(* Logix 5000 project; controller TBEN_Lx_8IOL_AOI_V0_1 vendor 1 type 14 code 176 rev 32.11; software revision 32.00; part 7 of 11 *)

TYPE Generic_131_Words :
STRUCT
   Data : INT[131];
END_STRUCT
END_TYPE

TYPE Generic_160_SINT :
STRUCT
   DATA : SINT[160];
END_STRUCT
END_TYPE

TYPE Generic_173_Words :
STRUCT
   Data : INT[173];
END_STRUCT
END_TYPE

TYPE Generic_5_Words :
STRUCT
   Data : INT[5];
END_STRUCT
END_TYPE

TYPE IOLRequest :
STRUCT
   Enable_Multiple_Nodes : BOOL;   // Set to 1 to enable multiple nodes
   ApplicationPath : STRING;   // Set Path for following IOL Instructions
   Read : BOOL;   // For internal use to integrate IOLRead and IOWrite with IOLService
   Write : BOOL;   // For internal use to integrate IOLRead and IOWrite with IOLService
   Reset : BOOL;   // For internal use to integrate IOLRead and IOWrite with IOLService
   Done : BOOL;   // For internal use to integrate IOLRead and IOWrite with IOLService
   Error : BOOL;   // For internal use to integrate IOLRead and IOWrite with IOLService
   Slot : INT;   // For internal use to integrate IOLRead and IOWrite with IOLService
   Port : INT;   // For internal use to integrate IOLRead and IOWrite with IOLService
   Index : INT;   // For internal use to integrate IOLRead and IOWrite with IOLService
   SubIndex : INT;   // For internal use to integrate IOLRead and IOWrite with IOLService
   Length : INT;   // For internal use to integrate IOLRead and IOWrite with IOLService
   Handle : INT;   // For internal use to integrate IOLRead and IOWrite with IOLService
   Status : INT;   // For internal use to integrate IOLRead and IOWrite with IOLService
   NextHandle : INT;   // For internal use to integrate IOLRead and IOWrite with IOLService
   ReceiveData : SINT[145];   // For internal use to integrate IOLRead and IOWrite with IOLService
   SendData : SINT[145];   // For internal use to integrate IOLRead and IOWrite with IOLService
   WriteData : DINT;   // For internal use to integrate IOLRead and IOWrite with IOLService
   ActivePath : STRING;   // For internal use to integrate IOLRead and IOWrite with IOLService
END_STRUCT
END_TYPE

TYPE Turck_IOLink_Common_Data :
STRUCT
   Read : BOOL;   // For internal use to integrate IOLRead and IOWrite with IOLService
   Write : BOOL;   // For internal use to integrate IOLRead and IOWrite with IOLService
   Reset : BOOL;   // For internal use to integrate IOLRead and IOWrite with IOLService
   Done : BOOL;   // For internal use to integrate IOLRead and IOWrite with IOLService
   Error : BOOL;   // For internal use to integrate IOLRead and IOWrite with IOLService
   Port_in_Use : SINT;   // Each bit is set to show that a port is in use. If it's not in use the port diagnostics will be disabled so IO-Link can still be used but won't throw a red light if no device plugged
   Port : INT;   // For internal use to integrate IOLRead and IOWrite with IOLService
   Index : INT;   // For internal use to integrate IOLRead and IOWrite with IOLService
   SubIndex : INT;   // For internal use to integrate IOLRead and IOWrite with IOLService
   Length : INT;   // For internal use to integrate IOLRead and IOWrite with IOLService
   TicketNum : INT;   // For internal use to integrate IOLRead and IOWrite with IOLService
   Status : INT;   // For internal use to integrate IOLRead and IOWrite with IOLService
   NextTicketNum : INT;   // For internal use to integrate IOLRead and IOWrite with IOLService
   Process_Input_Data : INT[128];
   Process_Output_Data : INT[128];
   ReceiveData : SINT[255];   // For internal use to integrate IOLRead and IOWrite with IOLService
   SendData : SINT[145];   // For internal use to integrate IOLRead and IOWrite with IOLService
   Vendor_IDs : INT[8];
   Device_IDs : DINT[8];
   WriteData : DINT;
END_STRUCT
END_TYPE

TYPE Universal_IOLink_Info :
STRUCT
   Vendor_Name : STRING;   // Index 16
   Vendor_Text : STRING;   // Index 17
   Product_Name : STRING;   // Index 18
   Product_ID : STRING;   // Index 19
   Product_Text : STRING;   // Index 20
   Serial_Number : STRING;   // Index 21
   Hardware_Revision : STRING;   // Index 22
   Firmware_Revision : STRING;   // Index 23
   Application_Specific_Tag : STRING;   // Index 24
   Function_Tag : STRING;   // Index 25
   Location_Tag : STRING;   // Index 26
   Application_Specific_Tag_Requested : STRING;
END_STRUCT
END_TYPE

ADD_ON_INSTRUCTION IOL_ReadData   (* revision 2.5 Support TBIP, ExecutePrescan, ExecuteEnableInFalse *)
// Revision note:
// V1_0 Initial Release
// V1_1 Automatic data precision detection
// V1_2 Added multiple EIP node support
// V2_5 Support TBIP
// Help:
// IOL_ReadData - used with Turck BL20, BL67, BLC and TBEN IOLink masters to read numeric data from IOLink devices.  Use in conjuction with IOLService AOI which processes all IOL read and write requests.
// Status	Description
// 0	Operation completed successfully
// 	Status = 100 - 102, Ethernet IP MSG instruction errors - check communication parameters
// 100	IOL_SendMSG completed with error, check communication parameters
// 101	IOL_RecevieMSG completed with error, check communication parameters
// 110	IOL_Service Retry Limit exceeded
// 111	Slot specified not an IOLink master
// 	Status = 1000 to 1255, no response from device, connection error
// 1016	Device not connected or Port not configured as IOLink port
// 	Status = 2000 to 2255,  device response indicates error
// 2000	Device error, no details
// 2017	Device error, Index not available
// 2018	Device error, Subindex not available
// 2032	Device error, Service temporarily not available
// 2033	Device error, Service temporarily not available - local control
// 2034	Device error, Service temporarily not available - device control
// 2035	Device error, Index not writeable
// 2048	Device error, Parameter value out of range
// 2049	Device error, Parameter value above limit
// 2050	Device error, Parameter value below limit
// 2051	Device error, Parameter value length overrun (check IOLWrite precision/string length)
// 2052	Device error, Parameter value length underrun (check IOLWrite precision/string length)
// 2053	Device error, Function not available
// 2054	Device error, Function temporarily not available
// 2064	Device error, Parameter set invalid
// 2065	Device error, Inconsistent parameter set
// 2130	Device error, Application not ready
// 	Status = 3000 to 3255,   device response indicates vendor specific error
// 3000	Vendor specific error, no details
// 3001	Vendor specific error, vendor specific error number
// 3255	Vendor specific error, vendor specific error number
// 	Status = 7000 to 7255,  IOL-M Error Codes
// 7000	Unexpected write request instead of read request
// 7001	Decode error
// 7002	Port occupied by another task
// 	Status = 8000 to 8255,  IOL-M Error Codes
// 8000	Timeout when IOL-Ds or IOL-M ports are busy
// 8001	IOL Index out of range
// 8002	Port address greater than maximum
// 8003	Port function not supported
VAR_OUTPUT
   Done : BOOL; {access Read Only, visible}   // IOLRead completed successfully
   Error : BOOL; {access Read Only, visible}   // IOLRead completed with error, check status
   Pending : BOOL; {access Read Only, visible}   // IOLRead waiting to be processed
   Active : BOOL; {access Read Only, visible}   // IOLRead in progress
END_VAR
VAR_IN_OUT
   Common_Data : IOLRequest; {required}   // Shared IOL Data Area - must be identical on all requests
END_VAR
VAR_OUTPUT
   DoneCount : DINT; {access Read Only, visible}   // Number of operations completed successfully
   ErrorCount : DINT; {access Read Only, visible}   // Number of operations competed with error
   Status : INT; {access Read Only, visible}   // Status of last IOLRead
END_VAR
VAR_INPUT
   Read : BOOL;   // Rising edge triggers IOLink Read
   Read_Continuous : BOOL;   // Set to trigger IOLink Read repeatedly
   Slot : INT; {visible}   // IOLink Master slot number
   Port : INT; {visible}   // IOLink Master Port number, 1,2,3 or 4
   Index : INT; {visible}   // IOL Index number
   SubIndex : INT; {visible}   // IOL Subindex number
END_VAR
VAR_OUTPUT
   ReadData : DINT; {access Read Only, required}   // Data returned from IOLink device
END_VAR
VAR_INPUT
   R_8_Bit : BOOL;   // Indicates data received is 8 bit precision
   R_16_Bit : BOOL;   // Indicates data received is 16 bit precision
   R_32_Bit : BOOL;   // Indicates data received is 32 bit precision
   R_Sign_Extend : BOOL;   // Set to extend 8/16 bit precision data sign bit
   R_Swap_16 : BOOL;   // 16-bit AB->BA, 32-bit ABCD->BADC
   R_Swap_32 : BOOL;   // 32-bit ABCD->DCBA
   R_Swap_All : BOOL;   // 32-bit ABCD->CDBA
END_VAR
VAR
   MyHandle : INT;
   StartupDone : BOOL; {access None}
   Pending_or_Active : BOOL; {access None}
   Read_ONS : BOOL; {access None}
   StartupCount : DINT; {access None}
   ReadSignBit : DINT; {access None}
   ReadRequest : BOOL; {access None}
END_VAR

ROUTINE EnableInFalse   (* ladder *)
END_ROUTINE

ROUTINE Logic   (* ladder *)
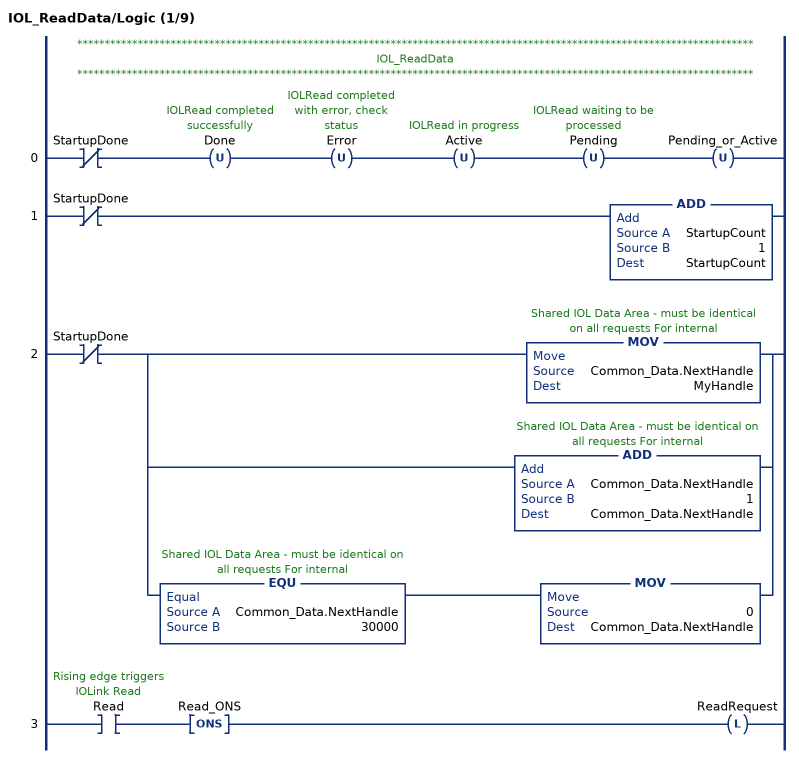
   // ***************************************************************************************************************************
   // IOL_ReadData
   // ***************************************************************************************************************************
   0: XIO(StartupDone)OTU(Done)OTU(Error)OTU(Active)OTU(Pending)OTU(Pending_or_Active);
   1: XIO(StartupDone)ADD(StartupCount,1,StartupCount);
   2: XIO(StartupDone)[MOV(Common_Data.NextHandle,MyHandle) ,ADD(Common_Data.NextHandle,1,Common_Data.NextHandle) ,EQU(Common_Data.NextHandle,30000) MOV(0,Common_Data.NextHandle) ];
   3: XIC(Read)ONS(Read_ONS)OTL(ReadRequest);
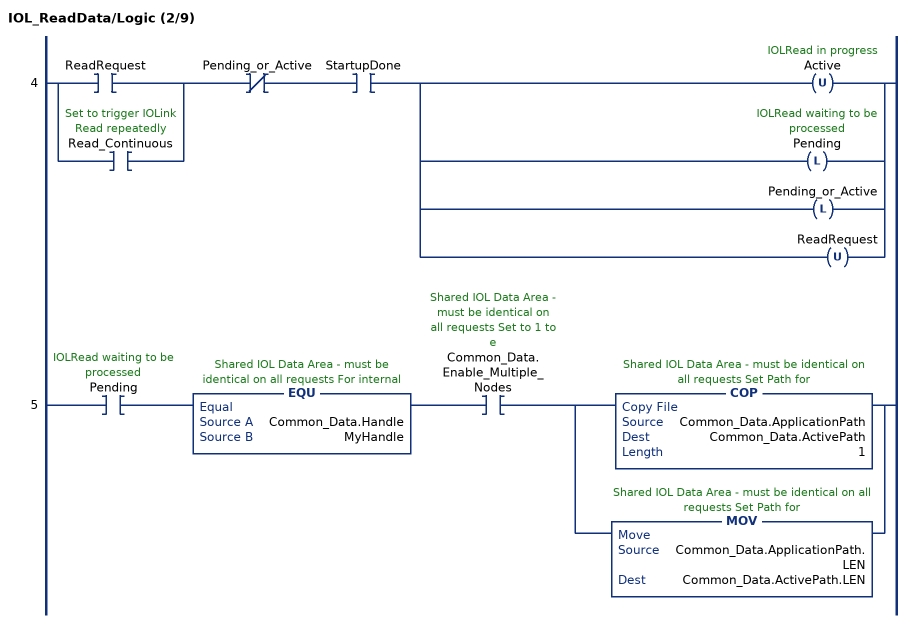
   4: [XIC(ReadRequest) ,XIC(Read_Continuous) ]XIO(Pending_or_Active)XIC(StartupDone)[OTU(Active) ,OTL(Pending) ,OTL(Pending_or_Active) ,OTU(ReadRequest) ];
   5: XIC(Pending)EQU(Common_Data.Handle,MyHandle)XIC(Common_Data.Enable_Multiple_Nodes)[COP(Common_Data.ApplicationPath,Common_Data.ActivePath,1) ,MOV(Common_Data.ApplicationPath.LEN,Common_Data.ActivePath.LEN) ];
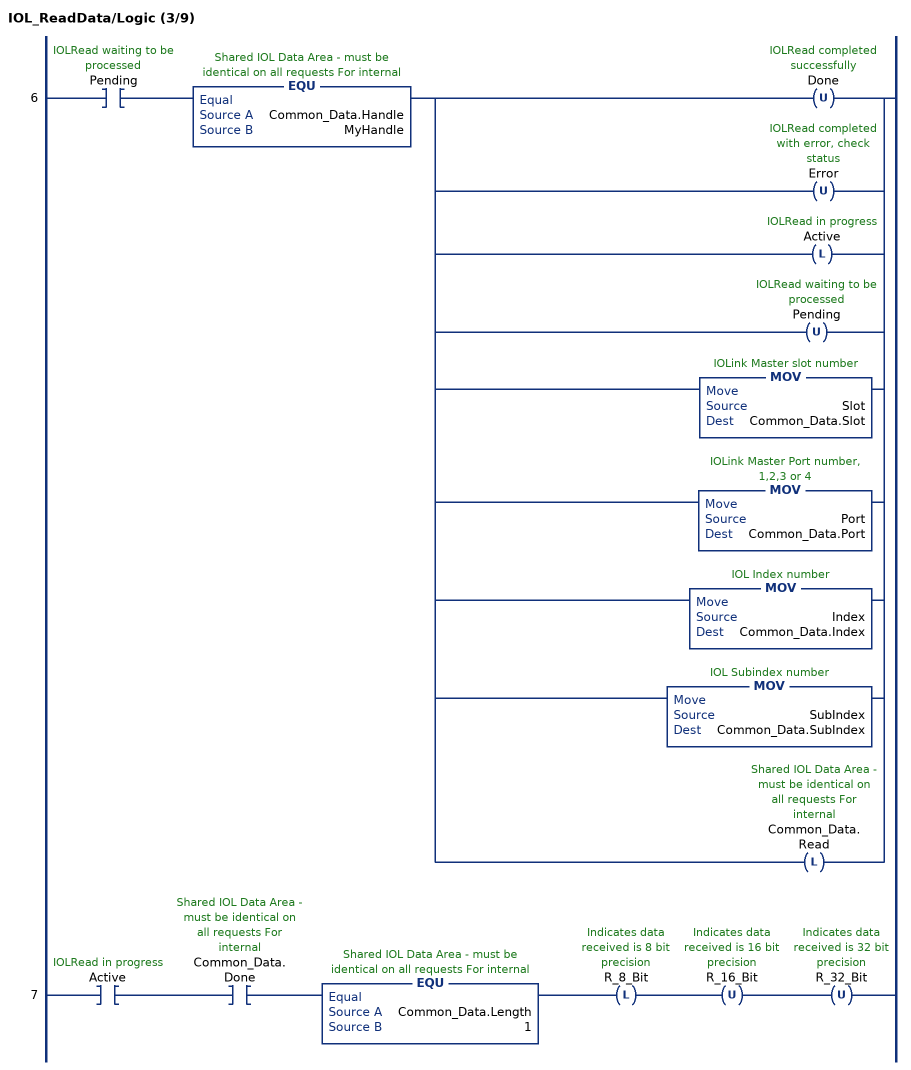
   6: XIC(Pending)EQU(Common_Data.Handle,MyHandle)[OTU(Done) ,OTU(Error) ,OTL(Active) ,OTU(Pending) ,MOV(Slot,Common_Data.Slot) ,MOV(Port,Common_Data.Port) ,MOV(Index,Common_Data.Index) ,MOV(SubIndex,Common_Data.SubIndex) ,OTL(Common_Data.Read) ];
   7: XIC(Active)XIC(Common_Data.Done)EQU(Common_Data.Length,1)OTL(R_8_Bit)OTU(R_16_Bit)OTU(R_32_Bit);
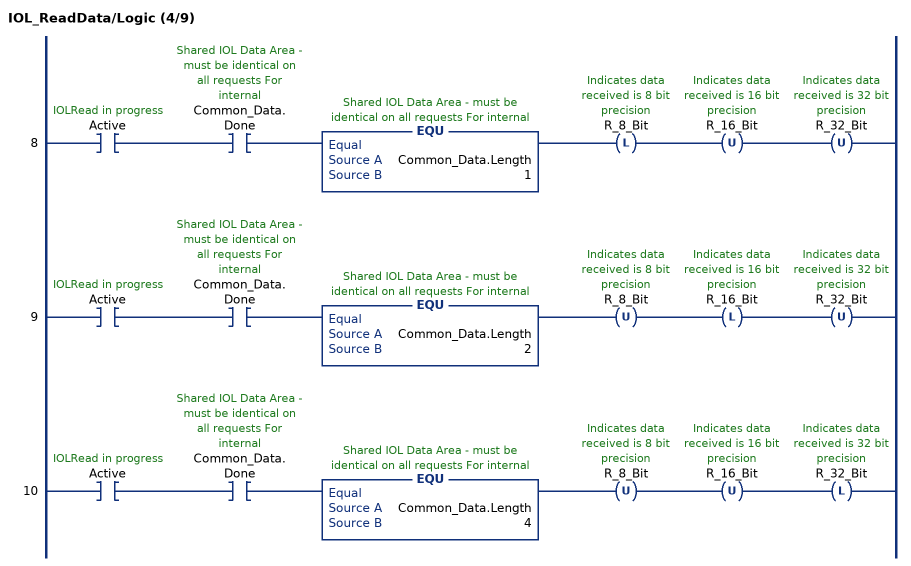
   8: XIC(Active)XIC(Common_Data.Done)EQU(Common_Data.Length,1)OTL(R_8_Bit)OTU(R_16_Bit)OTU(R_32_Bit);
   9: XIC(Active)XIC(Common_Data.Done)EQU(Common_Data.Length,2)OTU(R_8_Bit)OTL(R_16_Bit)OTU(R_32_Bit);
   10: XIC(Active)XIC(Common_Data.Done)EQU(Common_Data.Length,4)OTU(R_8_Bit)OTU(R_16_Bit)OTL(R_32_Bit);
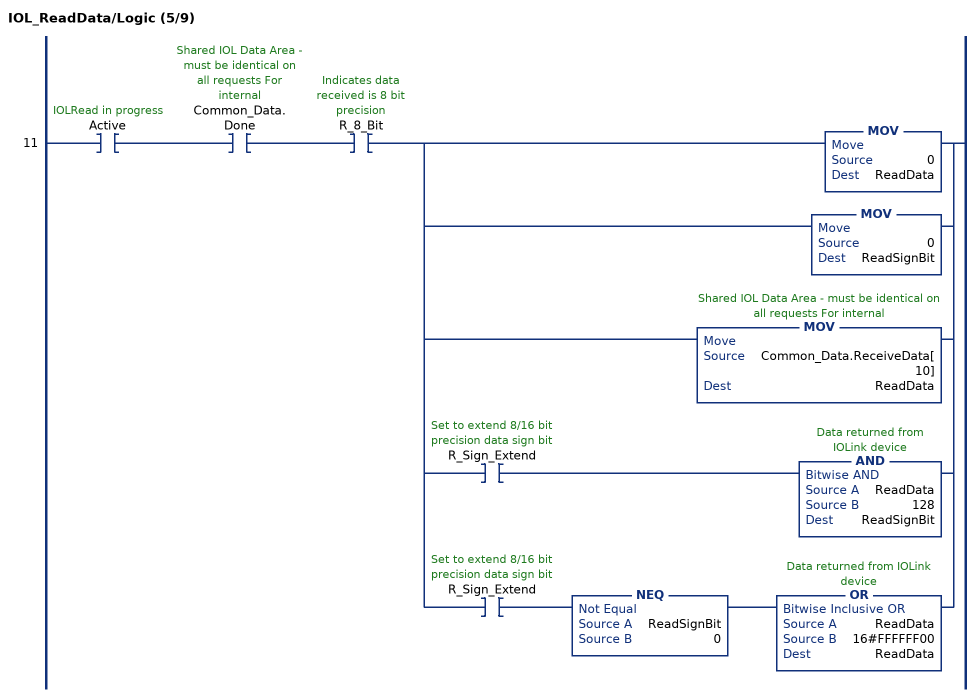
   11: XIC(Active)XIC(Common_Data.Done)XIC(R_8_Bit)[MOV(0,ReadData) ,MOV(0,ReadSignBit) ,MOV(Common_Data.ReceiveData[10],ReadData) ,XIC(R_Sign_Extend) AND(ReadData,128,ReadSignBit) ,XIC(R_Sign_Extend) NEQ(ReadSignBit,0) OR(ReadData,16#FFFFFF00,ReadData) ];
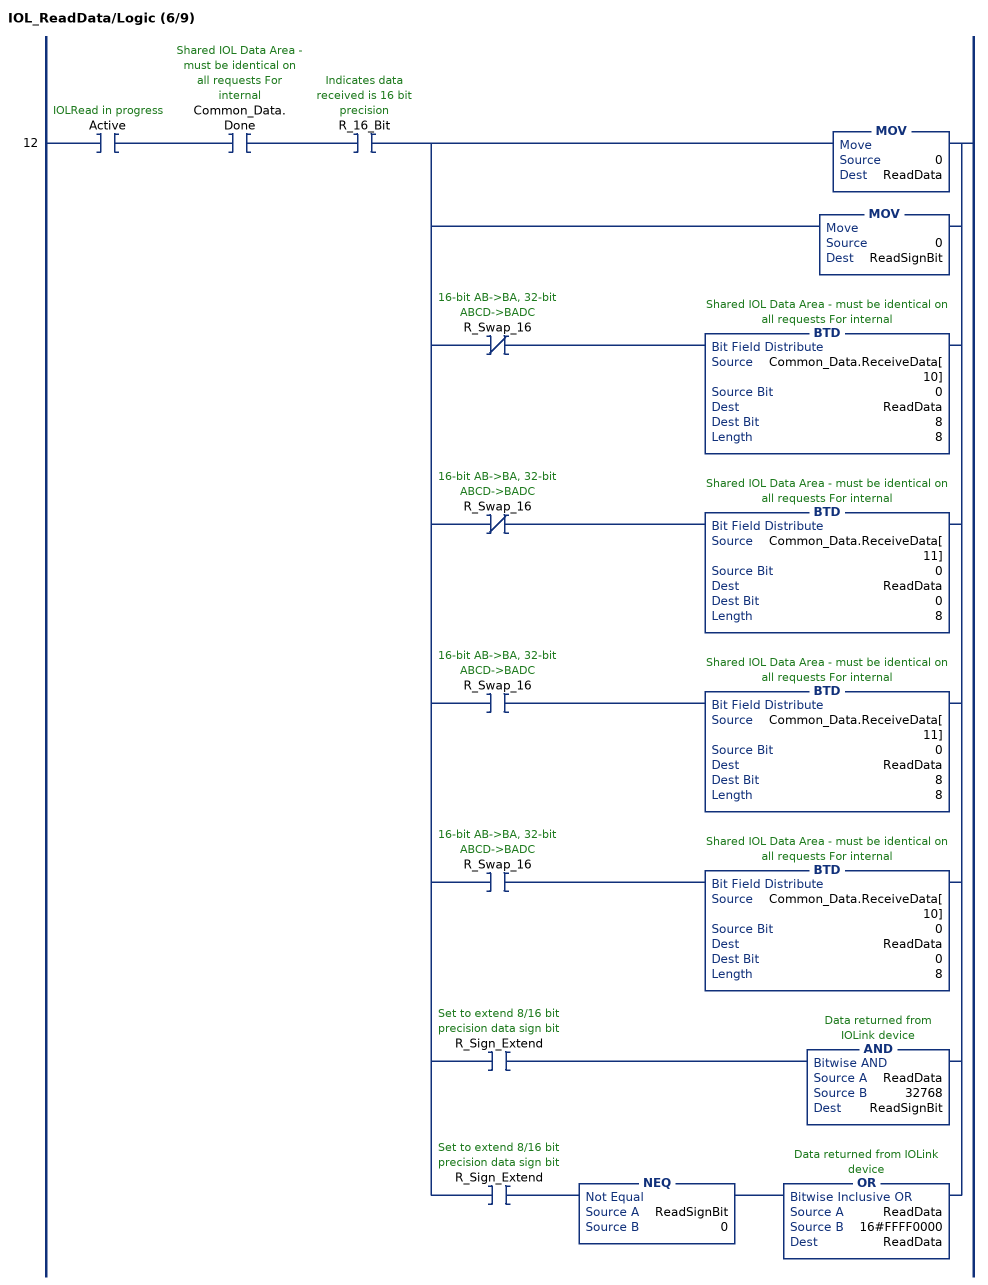
   12: XIC(Active)XIC(Common_Data.Done)XIC(R_16_Bit)[MOV(0,ReadData) ,MOV(0,ReadSignBit) ,XIO(R_Swap_16) BTD(Common_Data.ReceiveData[10],0,ReadData,8,8) ,XIO(R_Swap_16) BTD(Common_Data.ReceiveData[11],0,ReadData,0,8) ,XIC(R_Swap_16) BTD(Common_Data.ReceiveData[11],0,ReadData,8,8) ,XIC(R_Swap_16) BTD(Common_Data.ReceiveData[10],0,ReadData,0,8) ,XIC(R_Sign_Extend) AND(ReadData,32768,ReadSignBit) ,XIC(R_Sign_Extend) NEQ(ReadSignBit,0) OR(ReadData,16#FFFF0000,ReadData) ];
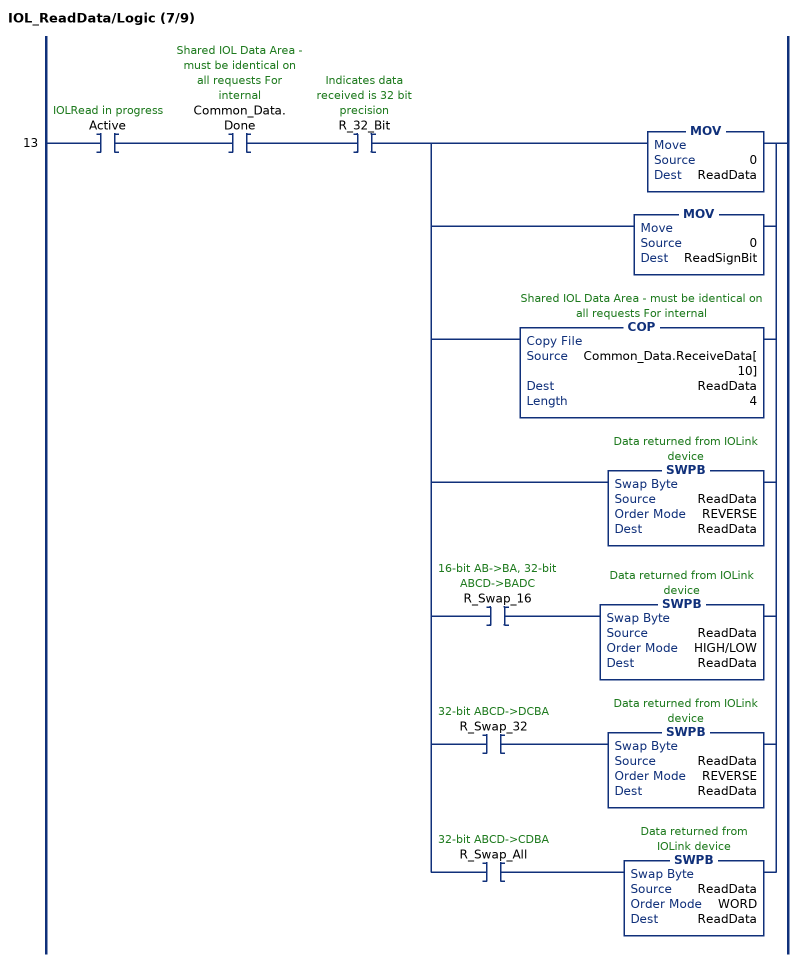
   13: XIC(Active)XIC(Common_Data.Done)XIC(R_32_Bit)[MOV(0,ReadData) ,MOV(0,ReadSignBit) ,COP(Common_Data.ReceiveData[10],ReadData,4) ,SWPB(ReadData,REVERSE,ReadData) ,XIC(R_Swap_16) SWPB(ReadData,HIGH/LOW,ReadData) ,XIC(R_Swap_32) SWPB(ReadData,REVERSE,ReadData) ,XIC(R_Swap_All) SWPB(ReadData,WORD,ReadData) ];
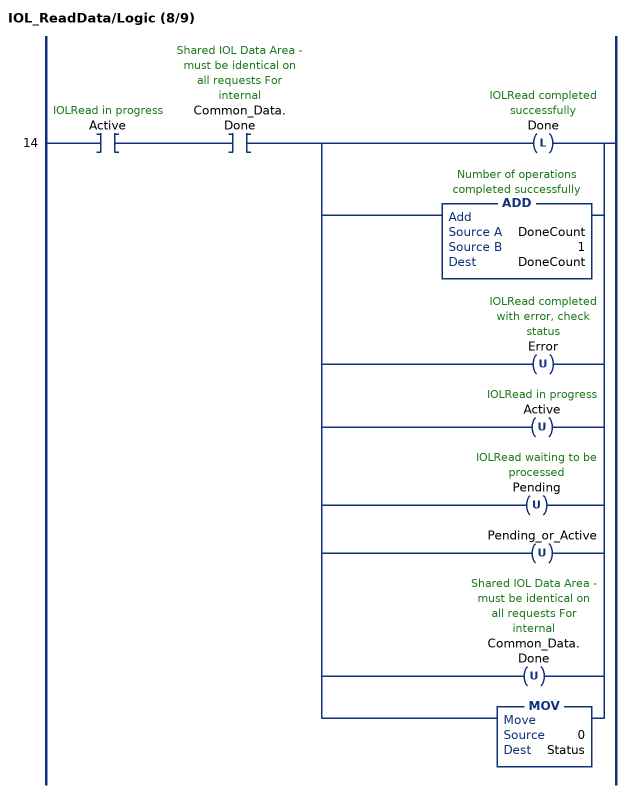
   14: XIC(Active)XIC(Common_Data.Done)[OTL(Done) ,ADD(DoneCount,1,DoneCount) ,OTU(Error) ,OTU(Active) ,OTU(Pending) ,OTU(Pending_or_Active) ,OTU(Common_Data.Done) ,MOV(0,Status) ];
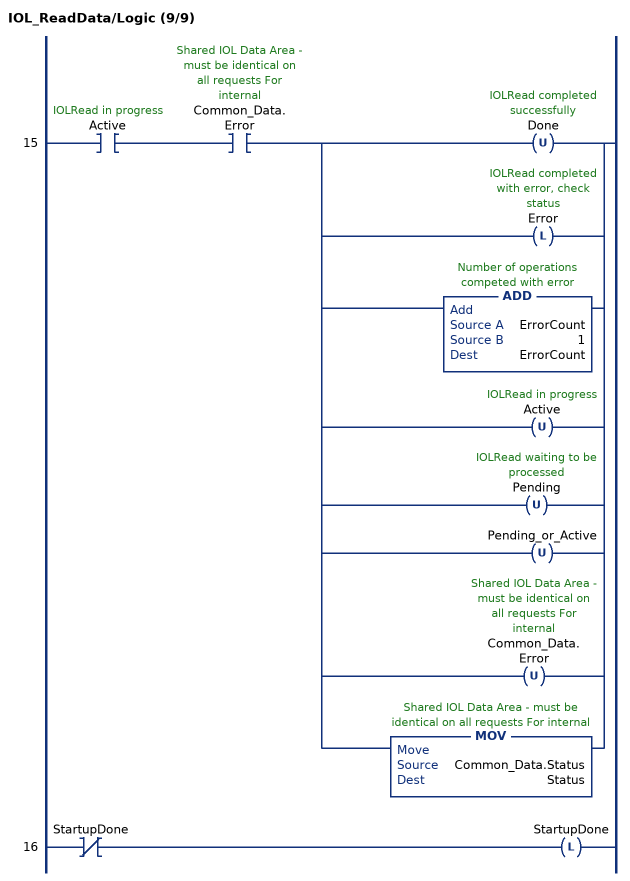
   15: XIC(Active)XIC(Common_Data.Error)[OTU(Done) ,OTL(Error) ,ADD(ErrorCount,1,ErrorCount) ,OTU(Active) ,OTU(Pending) ,OTU(Pending_or_Active) ,OTU(Common_Data.Error) ,MOV(Common_Data.Status,Status) ];
   16: XIO(StartupDone)OTL(StartupDone);
END_ROUTINE

ROUTINE Prescan   (* ladder *)
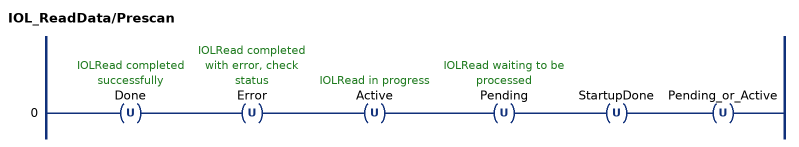
   0: OTU(Done)OTU(Error)OTU(Active)OTU(Pending)OTU(StartupDone)OTU(Pending_or_Active);
END_ROUTINE
END_ADD_ON_INSTRUCTION

ADD_ON_INSTRUCTION IOLService_ISDU   (* revision 1.0 Initial Release, ExecutePrescan *)
// Replace DSID with ISDU in Turck IOLC AOI interface
// KH 6/19/2023
// Revision note:
// V1_0 Initial Release
// Help:
// IOL_Service - used with Turck BL20, BL67, BLC and TBEN IOLink masters to process requests from IOL_ReadString, IOL_WriteString, IOL_ReadData and IOL_WriteData AOI's.
// Status	Description
// 0	Operation completed successfully
// 	Status = 100 - 102, Ethernet IP MSG instruction errors - check communication parameters
// 100	IOL_SendMSG completed with error, check communication parameters
// 101	IOL_RecevieMSG completed with error, check communication parameters
// 110	IOL_Service Retry Limit exceeded
// 111	Slot specified not an IOLink master
// 	Status = 1000 to 1255, no response from device, connection error
// 1016	Device not connected or Port not configured as IOLink port
// 	Status = 2000 to 2255,  device response indicates error
// 2000	Device error, no details
// 2017	Device error, Index not available
// 2018	Device error, Subindex not available
// 2032	Device error, Service temporarily not available
// 2033	Device error, Service temporarily not available - local control
// 2034	Device error, Service temporarily not available - device control
// 2035	Device error, Index not writeable
// 2048	Device error, Parameter value out of range
// 2049	Device error, Parameter value above limit
// 2050	Device error, Parameter value below limit
// 2051	Device error, Parameter value length overrun (check IOLWrite precision/string length)
// 2052	Device error, Parameter value length underrun (check IOLWrite precision/string length)
// 2053	Device error, Function not available
// 2054	Device error, Function temporarily not available
// 2064	Device error, Parameter set invalid
// 2065	Device error, Inconsistent parameter set
// 2130	Device error, Application not ready
// 	Status = 3000 to 3255,   device response indicates vendor specific error
// 3000	Vendor specific error, no details
// 3001	Vendor specific error, vendor specific error number
// 3255	Vendor specific error, vendor specific error number
// 	Status = 7000 to 7255,  IOL-M Error Codes
// 7000	Unexpected write request instead of read request
// 7001	Decode error
// 7002	Port occupied by another task
// 	Status = 8000 to 8255,  IOL-M Error Codes
// 8000	Timeout when IOL-Ds or IOL-M ports are busy
// 8001	IOL Index out of range
// 8002	Port address greater than maximum
// 8003	Port function not supported
VAR_IN_OUT
   Common_Data : Turck_IOLink_Common_Data; {required}
        .SendData[1]   // For internal use to integrate IOLRead and IOLWrite with IOLService
   IOL_Read_MSG : MESSAGE; {required}
   IOL_Write_MSG : MESSAGE; {required}
   Process_Input_Data : Generic_173_Words; {required}
   Process_Output_Data : Generic_131_Words; {required}
END_VAR
VAR
   IOLReadActive : BOOL;
   IOLWriteActive : BOOL;
   RetryCount : DINT;
   IOL_Error_Count : DINT; {access None}
   IOLReset_ONS : BOOL; {access None}
   ER1 : BOOL; {access None}
   ER2 : BOOL; {access None}
   tempReceiveData : SINT[255]; {access None}
   Generate_Status : BOOL; {access None}
   ABS_RD_0 : INT; {access None}
   ABS_RD_1 : INT; {access None}
   ABS_RD_2 : INT; {access None}
   ABS_RD_3 : INT; {access None}
   tempSendData : SINT[145]; {access None}
   IOL_READ_Request : BOOL; {access None}
   IOL_WRITE_Request : BOOL; {access None}
   StartupDone : BOOL; {access None}
   Done : BOOL; {access None}
   Error : BOOL; {access None}
   Active : BOOL; {access None}
   Pending : BOOL; {access None}
   Pending_or_Active : BOOL; {access None}
   StartupCount : SINT; {access None}
   DoneCount : SINT; {access None}
   MyTicketNum : INT; {access None}
   Update_Data : BOOL; {access None}
   Read_ONS : BOOL; {access None}
   ReadRequest : BOOL; {access None}
   Prev_Input_Data_Valids : INT; {access None}
   Status : DINT; {access None}
   ErrorCount : DINT; {access None}
   PIDV_Delay : TIMER := (PRE := 1000); {access None}
END_VAR

ROUTINE Logic   (* ladder *)
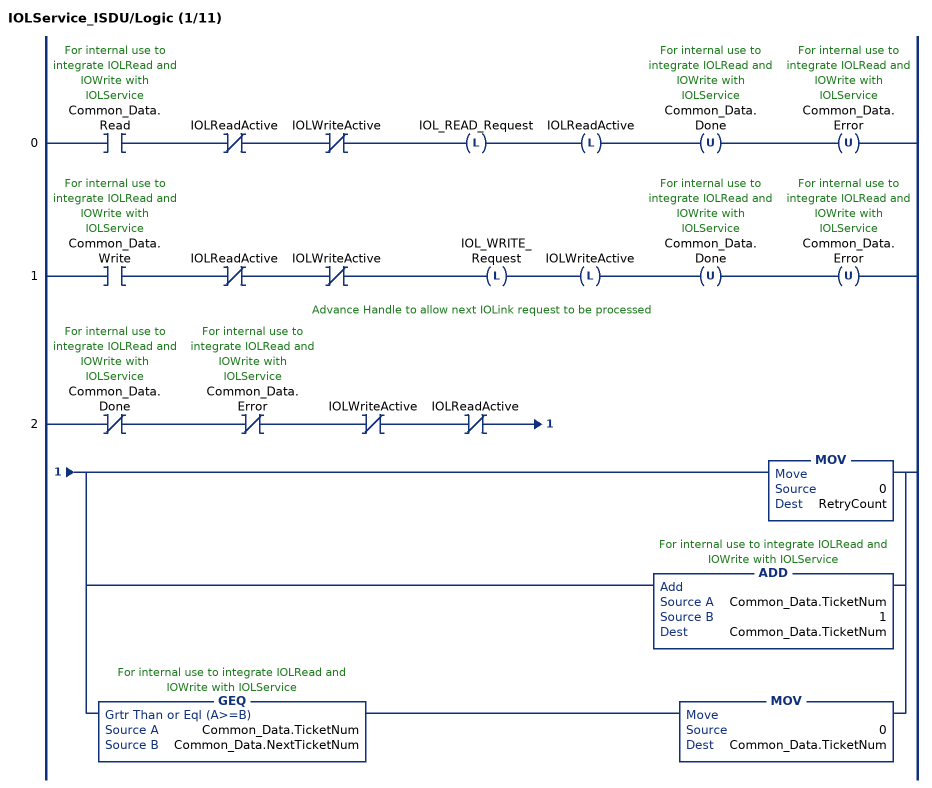
   0: XIC(Common_Data.Read)XIO(IOLReadActive)XIO(IOLWriteActive)OTL(IOL_READ_Request)OTL(IOLReadActive)OTU(Common_Data.Done)OTU(Common_Data.Error);
   1: XIC(Common_Data.Write)XIO(IOLReadActive)XIO(IOLWriteActive)OTL(IOL_WRITE_Request)OTL(IOLWriteActive)OTU(Common_Data.Done)OTU(Common_Data.Error);
   // Advance Handle to allow next IOLink request to be processed
   2: XIO(Common_Data.Done)XIO(Common_Data.Error)XIO(IOLWriteActive)XIO(IOLReadActive)[MOV(0,RetryCount) ,ADD(Common_Data.TicketNum,1,Common_Data.TicketNum) ,GEQ(Common_Data.TicketNum,Common_Data.NextTicketNum) MOV(0,Common_Data.TicketNum) ];
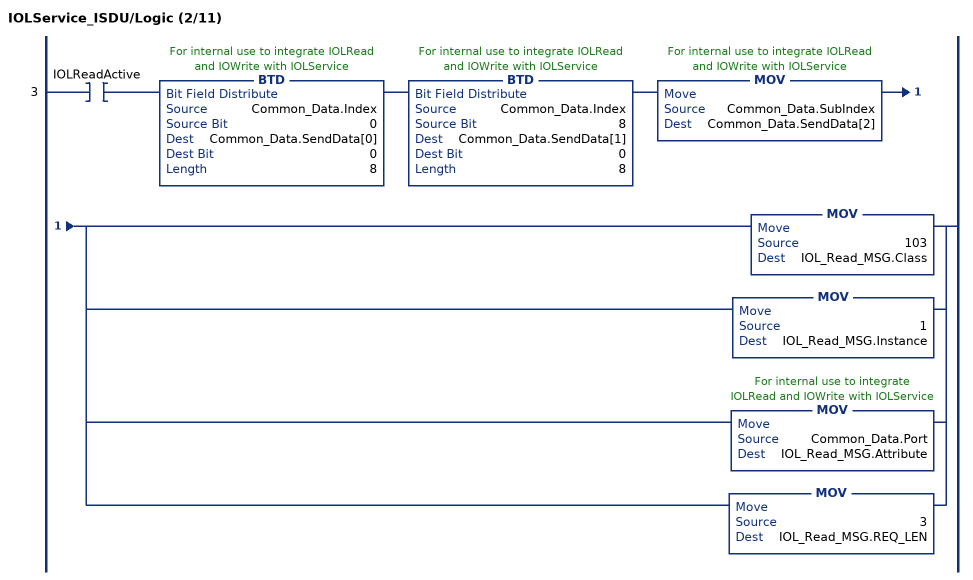
   3: XIC(IOLReadActive)BTD(Common_Data.Index,0,Common_Data.SendData[0],0,8)BTD(Common_Data.Index,8,Common_Data.SendData[1],0,8)MOV(Common_Data.SubIndex,Common_Data.SendData[2])[MOV(103,IOL_Read_MSG.Class) ,MOV(1,IOL_Read_MSG.Instance) ,MOV(Common_Data.Port,IOL_Read_MSG.Attribute) ,MOV(3,IOL_Read_MSG.REQ_LEN) ];
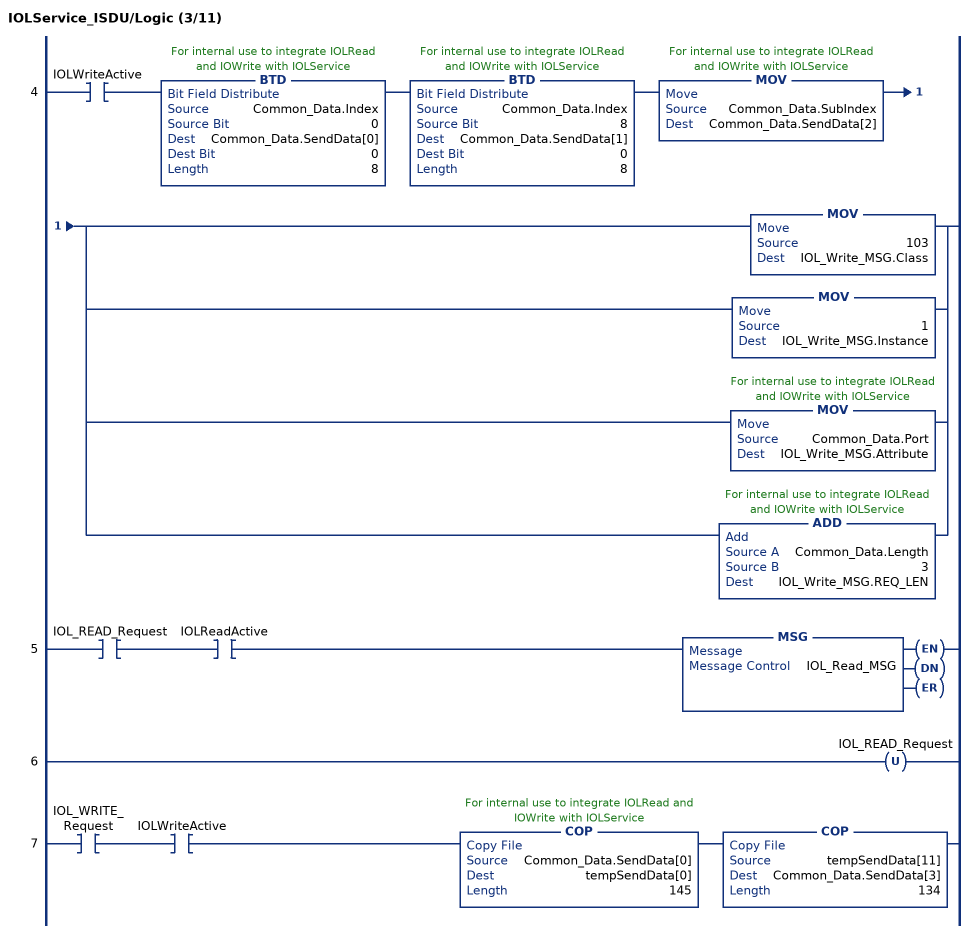
   4: XIC(IOLWriteActive)BTD(Common_Data.Index,0,Common_Data.SendData[0],0,8)BTD(Common_Data.Index,8,Common_Data.SendData[1],0,8)MOV(Common_Data.SubIndex,Common_Data.SendData[2])[MOV(103,IOL_Write_MSG.Class) ,MOV(1,IOL_Write_MSG.Instance) ,MOV(Common_Data.Port,IOL_Write_MSG.Attribute) ,ADD(Common_Data.Length,3,IOL_Write_MSG.REQ_LEN) ];
   5: XIC(IOL_READ_Request)XIC(IOLReadActive)MSG(IOL_Read_MSG);
   6: OTU(IOL_READ_Request);
   7: XIC(IOL_WRITE_Request)XIC(IOLWriteActive)COP(Common_Data.SendData[0],tempSendData[0],145)COP(tempSendData[11],Common_Data.SendData[3],134);
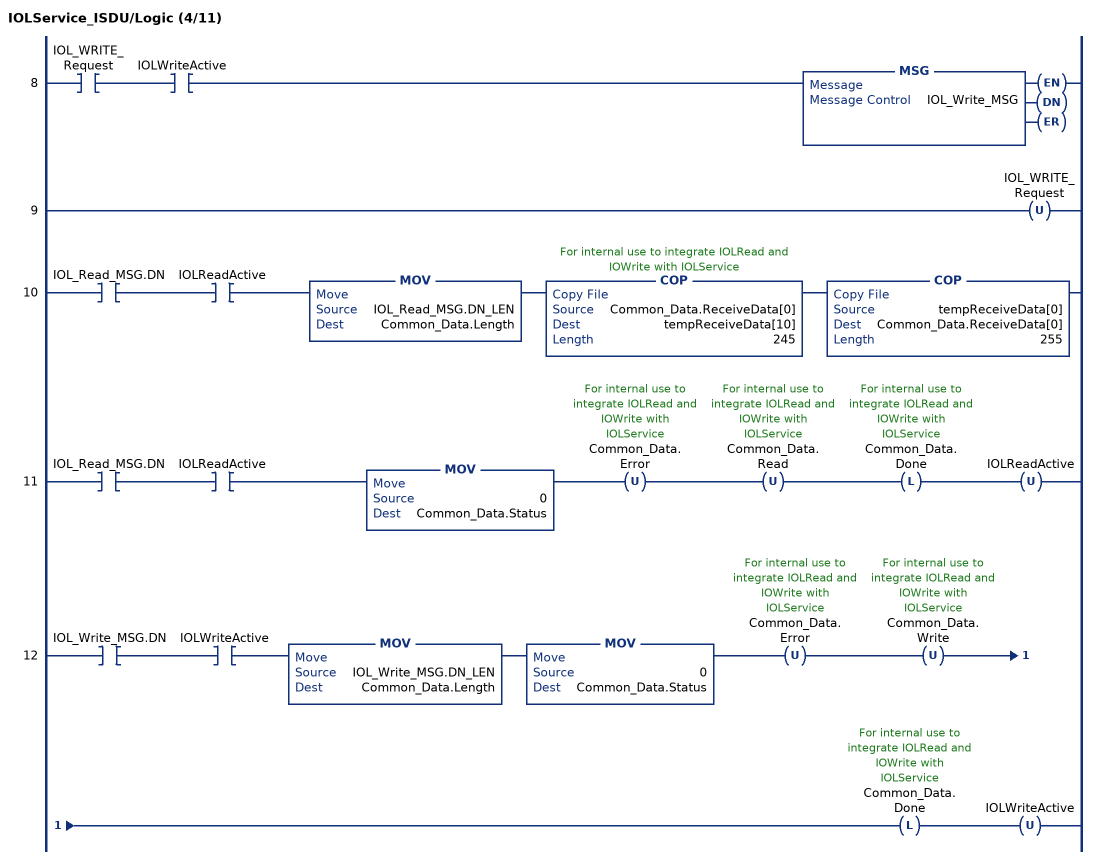
   8: XIC(IOL_WRITE_Request)XIC(IOLWriteActive)MSG(IOL_Write_MSG);
   9: OTU(IOL_WRITE_Request);
   10: XIC(IOL_Read_MSG.DN)XIC(IOLReadActive)MOV(IOL_Read_MSG.DN_LEN,Common_Data.Length)COP(Common_Data.ReceiveData[0],tempReceiveData[10],245)COP(tempReceiveData[0],Common_Data.ReceiveData[0],255);
   11: XIC(IOL_Read_MSG.DN)XIC(IOLReadActive)MOV(0,Common_Data.Status)OTU(Common_Data.Error)OTU(Common_Data.Read)OTL(Common_Data.Done)OTU(IOLReadActive);
   12: XIC(IOL_Write_MSG.DN)XIC(IOLWriteActive)MOV(IOL_Write_MSG.DN_LEN,Common_Data.Length)MOV(0,Common_Data.Status)OTU(Common_Data.Error)OTU(Common_Data.Write)OTL(Common_Data.Done)OTU(IOLWriteActive);
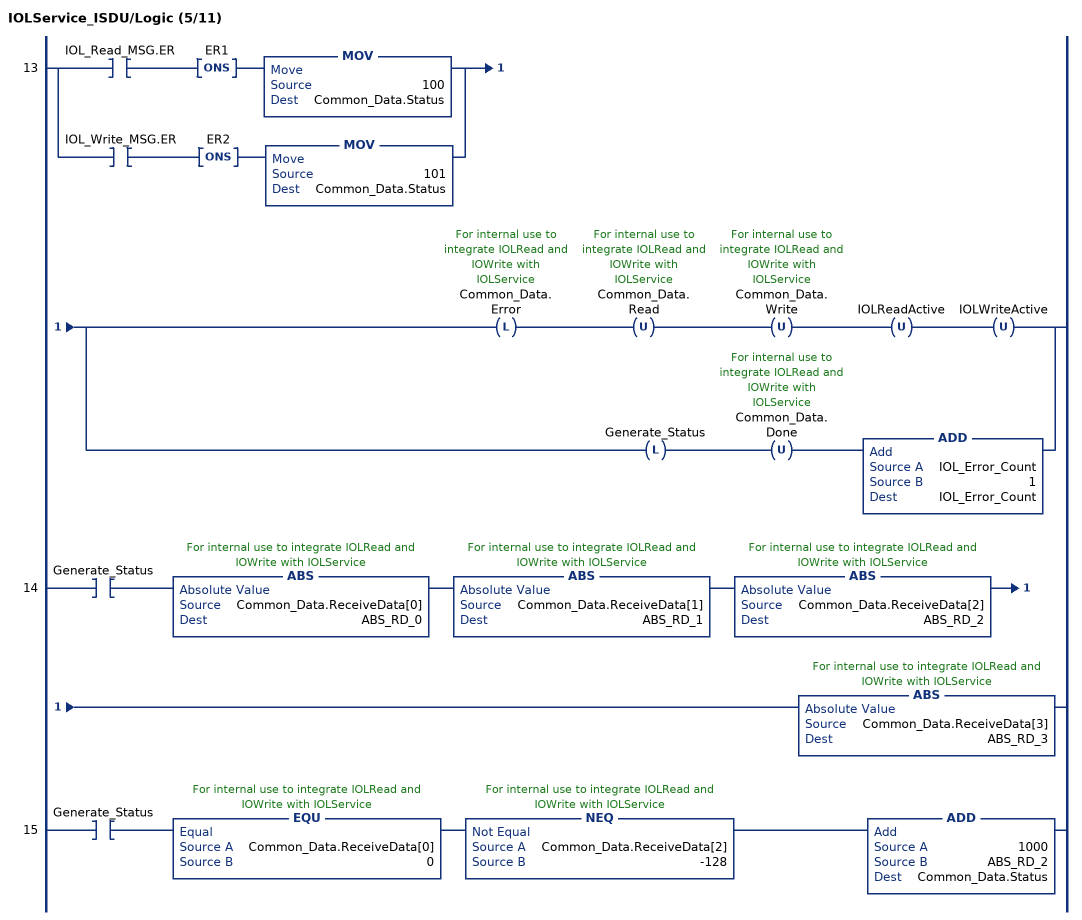
   13: [XIC(IOL_Read_MSG.ER) ONS(ER1) MOV(100,Common_Data.Status) ,XIC(IOL_Write_MSG.ER) ONS(ER2) MOV(101,Common_Data.Status) ][OTL(Common_Data.Error) OTU(Common_Data.Read) OTU(Common_Data.Write) OTU(IOLReadActive) OTU(IOLWriteActive) ,OTL(Generate_Status) OTU(Common_Data.Done) ADD(IOL_Error_Count,1,IOL_Error_Count) ];
   14: XIC(Generate_Status)ABS(Common_Data.ReceiveData[0],ABS_RD_0)ABS(Common_Data.ReceiveData[1],ABS_RD_1)ABS(Common_Data.ReceiveData[2],ABS_RD_2)ABS(Common_Data.ReceiveData[3],ABS_RD_3);
   15: XIC(Generate_Status)EQU(Common_Data.ReceiveData[0],0)NEQ(Common_Data.ReceiveData[2],-128)ADD(1000,ABS_RD_2,Common_Data.Status);
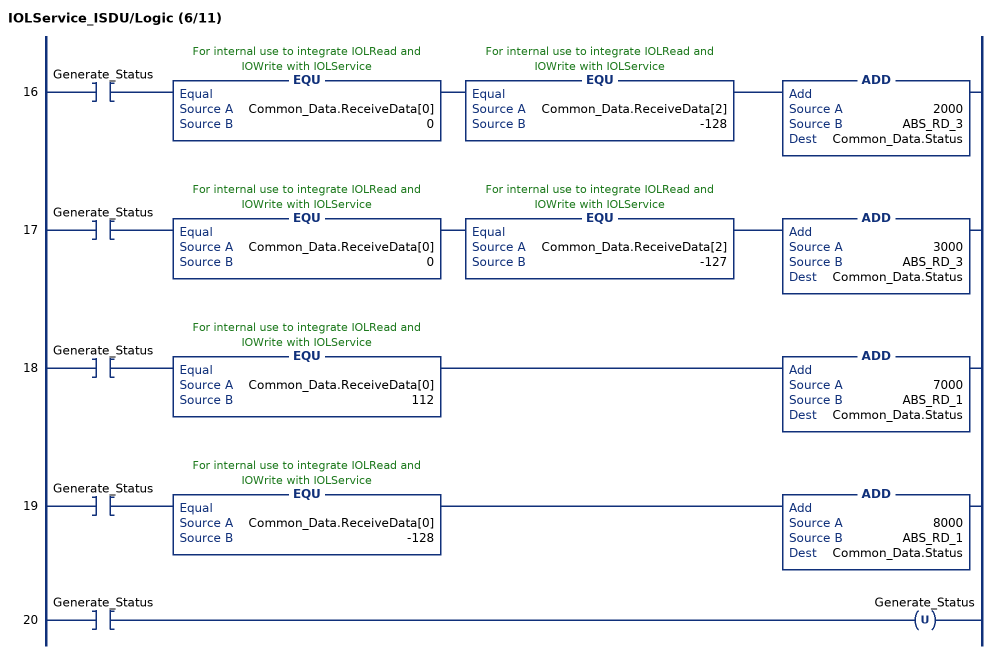
   16: XIC(Generate_Status)EQU(Common_Data.ReceiveData[0],0)EQU(Common_Data.ReceiveData[2],-128)ADD(2000,ABS_RD_3,Common_Data.Status);
   17: XIC(Generate_Status)EQU(Common_Data.ReceiveData[0],0)EQU(Common_Data.ReceiveData[2],-127)ADD(3000,ABS_RD_3,Common_Data.Status);
   18: XIC(Generate_Status)EQU(Common_Data.ReceiveData[0],112)ADD(7000,ABS_RD_1,Common_Data.Status);
   19: XIC(Generate_Status)EQU(Common_Data.ReceiveData[0],-128)ADD(8000,ABS_RD_1,Common_Data.Status);
   20: XIC(Generate_Status)OTU(Generate_Status);
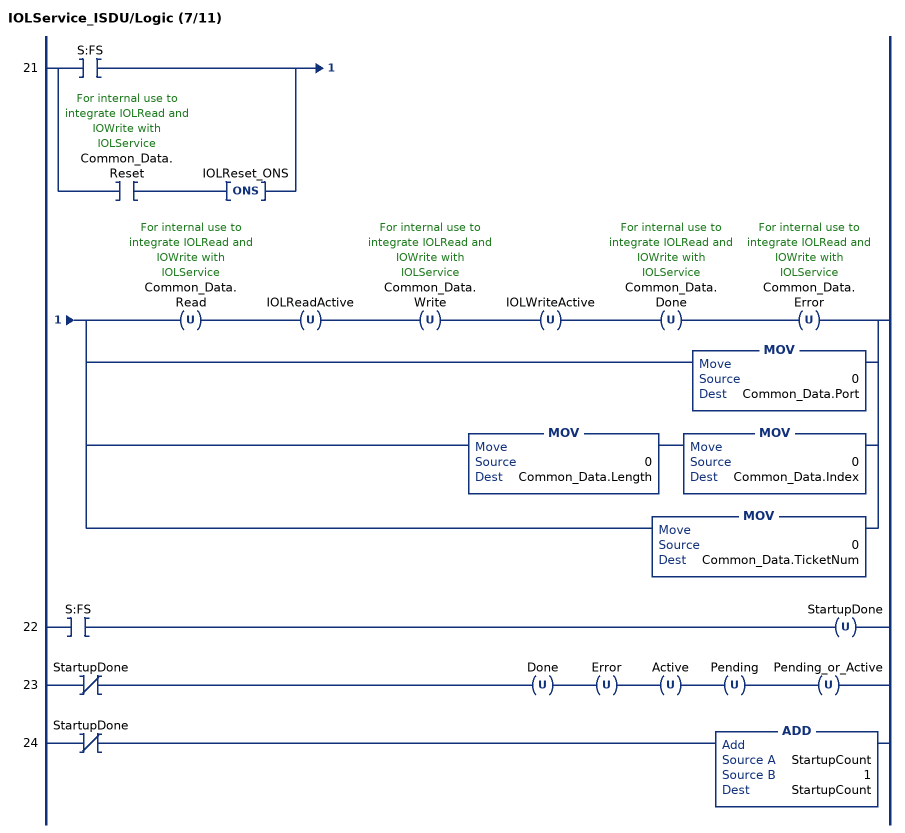
   21: [XIC(S:FS) ,XIC(Common_Data.Reset) ONS(IOLReset_ONS) ][OTU(Common_Data.Read) OTU(IOLReadActive) OTU(Common_Data.Write) OTU(IOLWriteActive) OTU(Common_Data.Done) OTU(Common_Data.Error) ,MOV(0,Common_Data.Port) ,MOV(0,Common_Data.Length) MOV(0,Common_Data.Index) ,MOV(0,Common_Data.TicketNum) ];
   22: XIC(S:FS)OTU(StartupDone);
   23: XIO(StartupDone)OTU(Done)OTU(Error)OTU(Active)OTU(Pending)OTU(Pending_or_Active);
   24: XIO(StartupDone)ADD(StartupCount,1,StartupCount);
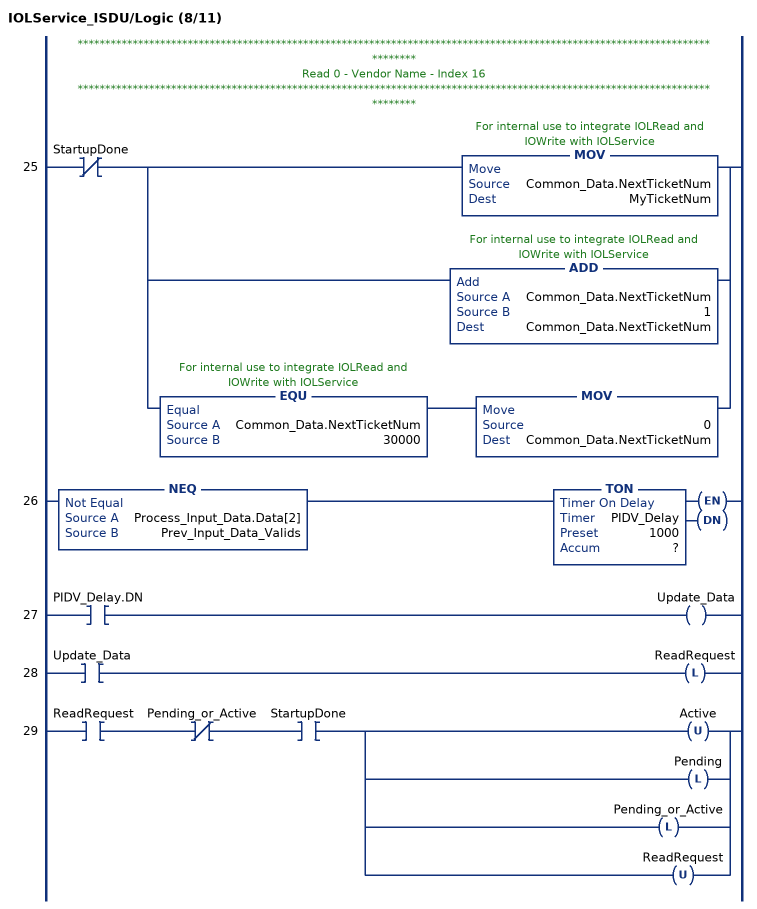
   // ***************************************************************************************************************************
   // Read 0 - Vendor Name - Index 16
   // ***************************************************************************************************************************
   25: XIO(StartupDone)[MOV(Common_Data.NextTicketNum,MyTicketNum) ,ADD(Common_Data.NextTicketNum,1,Common_Data.NextTicketNum) ,EQU(Common_Data.NextTicketNum,30000) MOV(0,Common_Data.NextTicketNum) ];
   26: NEQ(Process_Input_Data.Data[2],Prev_Input_Data_Valids)TON(PIDV_Delay,?,?);
   27: XIC(PIDV_Delay.DN)OTE(Update_Data);
   28: XIC(Update_Data)OTL(ReadRequest);
   29: XIC(ReadRequest)XIO(Pending_or_Active)XIC(StartupDone)[OTU(Active) ,OTL(Pending) ,OTL(Pending_or_Active) ,OTU(ReadRequest) ];
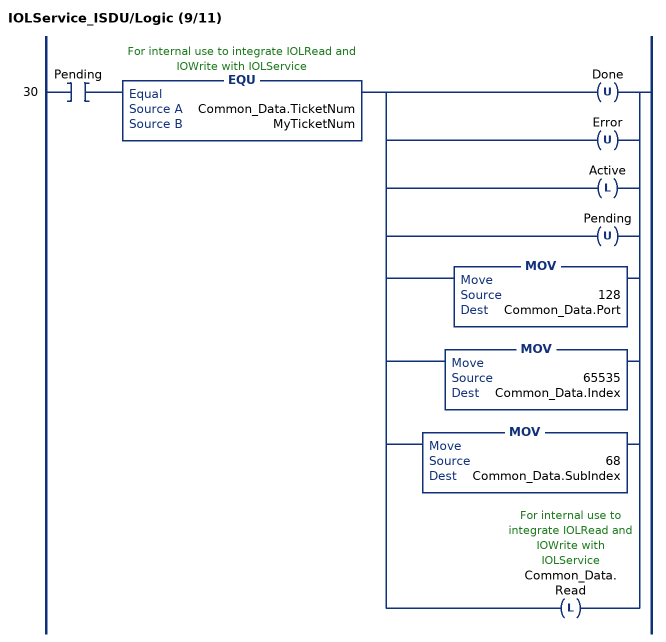
   30: XIC(Pending)EQU(Common_Data.TicketNum,MyTicketNum)[OTU(Done) ,OTU(Error) ,OTL(Active) ,OTU(Pending) ,MOV(128,Common_Data.Port) ,MOV(65535,Common_Data.Index) ,MOV(68,Common_Data.SubIndex) ,OTL(Common_Data.Read) ];
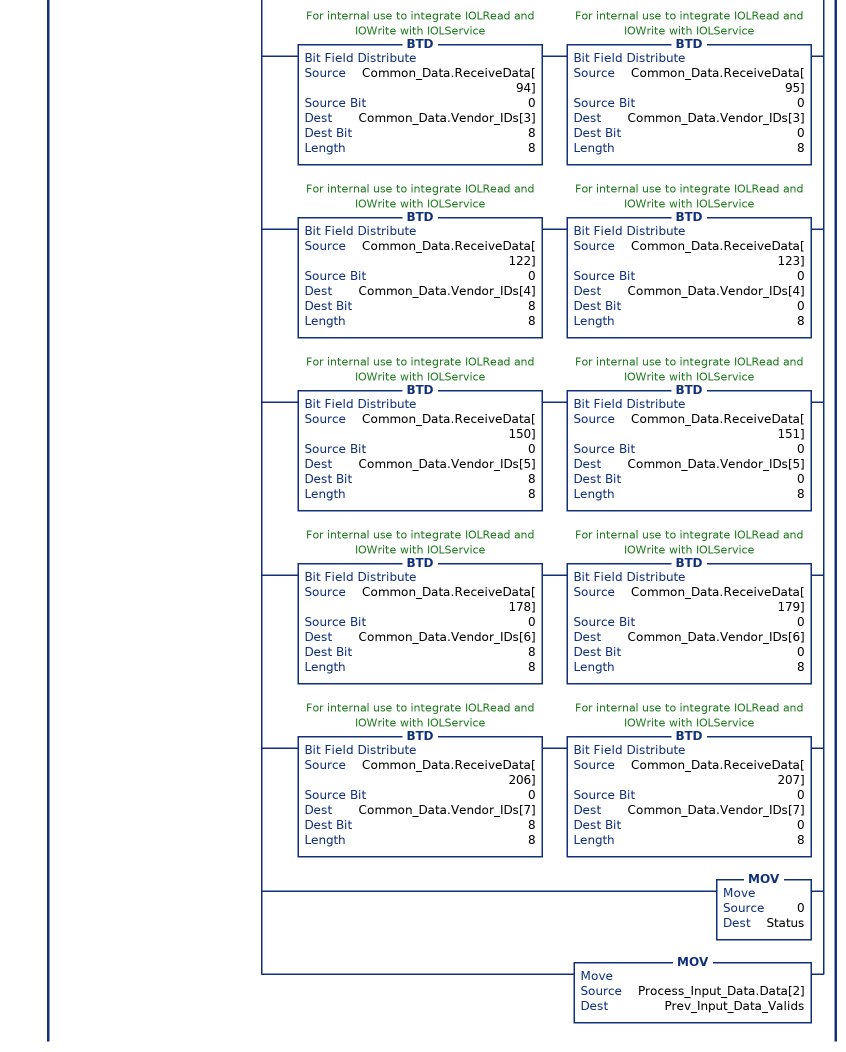
   31: XIC(Active)XIC(Common_Data.Done)[OTL(Done) ,ADD(DoneCount,1,DoneCount) ,OTU(Error) ,OTU(Active) ,OTU(Pending) ,OTU(Pending_or_Active) ,OTU(Common_Data.Done) ,BTD(Common_Data.ReceiveData[10],0,Common_Data.Vendor_IDs[0],8,8) BTD(Common_Data.ReceiveData[11],0,Common_Data.Vendor_IDs[0],0,8) ,BTD(Common_Data.ReceiveData[38],0,Common_Data.Vendor_IDs[1],8,8) BTD(Common_Data.ReceiveData[39],0,Common_Data.Vendor_IDs[1],0,8) ,BTD(Common_Data.ReceiveData[66],0,Common_Data.Vendor_IDs[2],8,8) BTD(Common_Data.ReceiveData[67],0,Common_Data.Vendor_IDs[2],0,8) ,BTD(Common_Data.ReceiveData[94],0,Common_Data.Vendor_IDs[3],8,8) BTD(Common_Data.ReceiveData[95],0,Common_Data.Vendor_IDs[3],0,8) ,BTD(Common_Data.ReceiveData[122],0,Common_Data.Vendor_IDs[4],8,8) BTD(Common_Data.ReceiveData[123],0,Common_Data.Vendor_IDs[4],0,8) ,BTD(Common_Data.ReceiveData[150],0,Common_Data.Vendor_IDs[5],8,8) BTD(Common_Data.ReceiveData[151],0,Common_Data.Vendor_IDs[5],0,8) ,BTD(Common_Data.ReceiveData[178],0,Common_Data.Vendor_IDs[6],8,8) BTD(Common_Data.ReceiveData[179],0,Common_Data.Vendor_IDs[6],0,8) ,BTD(Common_Data.ReceiveData[206],0,Common_Data.Vendor_IDs[7],8,8) BTD(Common_Data.ReceiveData[207],0,Common_Data.Vendor_IDs[7],0,8) ,MOV(0,Status) ,MOV(Process_Input_Data.Data[2],Prev_Input_Data_Valids) ];
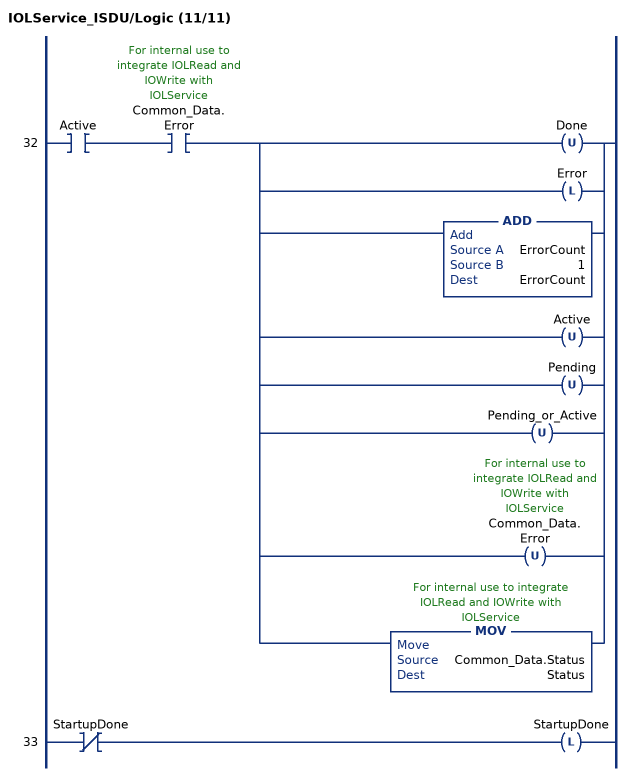
   32: XIC(Active)XIC(Common_Data.Error)[OTU(Done) ,OTL(Error) ,ADD(ErrorCount,1,ErrorCount) ,OTU(Active) ,OTU(Pending) ,OTU(Pending_or_Active) ,OTU(Common_Data.Error) ,MOV(Common_Data.Status,Status) ];
   33: XIO(StartupDone)OTL(StartupDone);
END_ROUTINE
